(* IEC 61131-3 sources: xPLCCore/codesys_code/Application/COMM_FBs/FB_MsgPakLevelParser, 7 files *)

(* ---- FB_MsgPakLevelParser.st ---- *)
(* ============================================================================
   FB_MsgPakLevelParser

   A state machine-based parser for MessagePack packets that processes data
   byte-by-byte and tracks the nesting level/depth of containers (arrays and maps).

   This parser does NOT decode MessagePack values, only tracks structure depth.
   ============================================================================ *)

FUNCTION_BLOCK FB_MsgPakLevelParser
VAR_INPUT
    in_byte : BYTE;  (* The byte to parse. Call this FB with a new byte for each step. *)
    x_reset : BOOL;  (* Set TRUE to reset the parser state. *)
END_VAR

VAR_OUTPUT
    stk_level_stack : ARRAY[0..29] OF UDINT;  (* Level stack showing remaining elements at each nesting level *)
    ui_level_stack_size : UDINT;              (* Current depth of the stack (number of nested containers) *)
    e_error : E_MsgPakLevelParser_ERROR;      (* Current error code (NONE if no error) *)
END_VAR

VAR
    (* State machine state *)
    e_state : E_MsgPakLevelParser_STATE;

    (* Length accumulation for variable-length types *)
    ui_length_bytes_remaining : UDINT;  (* How many length bytes still needed *)
    ui_length_value : UDINT;             (* Accumulated length value *)
    ui_data_bytes_remaining : UDINT;    (* How many data bytes still needed *)

    (* Track the type byte that caused us to enter EXPECT_LENGTH state *)
    by_last_type_byte : BYTE;  (* Last MessagePack type byte processed *)

    (* Constants *)
    c_MSGPACK_STACK_SIZE : UDINT := 30;  (* Maximum nesting depth *)

    (* Temporary variables *)
    by_current_byte : BYTE;
END_VAR
(* =========== IMPLEMENTATION =========== *)
(* ============================================================================
   Main State Machine Logic
   ============================================================================ *)

(* Handle reset *)
IF x_reset THEN
    ResetParser();
    RETURN;
END_IF

(* If error already occurred, stop processing *)
IF e_error <> E_MsgPakLevelParser_ERROR.NONE THEN
    RETURN;
END_IF

by_current_byte := in_byte;

CASE e_state OF
    E_MsgPakLevelParser_STATE.EXPECT_HEADER:
        (* Process MessagePack type byte *)
        HandleHeaderByte();

    E_MsgPakLevelParser_STATE.EXPECT_LENGTH:
        (* Accumulate length bytes *)
        ProcessLengthBytes();

    E_MsgPakLevelParser_STATE.EXPECT_EXT_TYPE:
        (* Consume extension type byte - no action needed, just transition *)
        e_state := E_MsgPakLevelParser_STATE.EXPECT_DATA;

    E_MsgPakLevelParser_STATE.EXPECT_DATA:
        (* Consume data bytes *)
        ProcessDataBytes();

    ELSE
        e_error := E_MsgPakLevelParser_ERROR.INVALID_STATE;
END_CASE

(* ---- DecrementStack.st ---- *)
METHOD DecrementStack : BOOL
VAR_INPUT
END_VAR
(* =========== IMPLEMENTATION =========== *)

(* Recursively decrement and pop completed levels *)
WHILE ui_level_stack_size > 0 DO
    (* Decrement current level *)
    IF stk_level_stack[ui_level_stack_size - 1] > 0 THEN
        stk_level_stack[ui_level_stack_size - 1] := stk_level_stack[ui_level_stack_size - 1] - 1;
    END_IF

    (* If items still remain in this container, we are done *)
    IF stk_level_stack[ui_level_stack_size - 1] > 0 THEN
        EXIT;
    END_IF

    (* If zero, pop this level and continue to decrement parent *)
    ui_level_stack_size := ui_level_stack_size - 1;
END_WHILE

(* ---- HandleHeaderByte.st ---- *)
METHOD HandleHeaderByte : INT
VAR_INPUT
END_VAR
VAR
    by_type : BYTE;
    ui_count : UDINT;
END_VAR
(* =========== IMPLEMENTATION =========== *)

by_type := by_current_byte;

(* Optimized: Check most common types first (FixInt covers ~50% of all values) *)
(* FixInt: positive (0x00-0x7F) and negative (0xE0-0xFF) *)
IF (by_type <= 16#7F) OR (by_type >= 16#E0) THEN
    DecrementStack();
    e_state := E_MsgPakLevelParser_STATE.EXPECT_HEADER;
    RETURN;
END_IF

(* FixMap (0x80-0x8F: 0-15 pairs) - common container type *)
IF (by_type >= 16#80) AND (by_type <= 16#8F) THEN
    ui_count := by_type - 16#80;
    IF ui_count > 0 THEN
        PushStack(ui_count * 2);
    ELSE
        DecrementStack();
    END_IF
    e_state := E_MsgPakLevelParser_STATE.EXPECT_HEADER;
    RETURN;
END_IF

(* FixArray (0x90-0x9F: 0-15 elements) - common container type *)
IF (by_type >= 16#90) AND (by_type <= 16#9F) THEN
    ui_count := by_type - 16#90;
    IF ui_count > 0 THEN
        PushStack(ui_count);
    ELSE
        DecrementStack();
    END_IF
    e_state := E_MsgPakLevelParser_STATE.EXPECT_HEADER;
    RETURN;
END_IF

(* FixStr (0xA0-0xBF: 0-31 bytes) - common string type *)
IF (by_type >= 16#A0) AND (by_type <= 16#BF) THEN
    ui_count := by_type - 16#A0;
    IF ui_count > 0 THEN
        ui_data_bytes_remaining := ui_count;
        e_state := E_MsgPakLevelParser_STATE.EXPECT_DATA;
    ELSE
        DecrementStack();
        e_state := E_MsgPakLevelParser_STATE.EXPECT_HEADER;
    END_IF
    RETURN;
END_IF

(* Use CASE for exact byte matches - more efficient than IF chain *)
CASE by_type OF
    16#C0:  (* nil *)
        DecrementStack();
        e_state := E_MsgPakLevelParser_STATE.EXPECT_HEADER;

    16#C2:  (* false *)
        DecrementStack();
        e_state := E_MsgPakLevelParser_STATE.EXPECT_HEADER;

    16#C3:  (* true *)
        DecrementStack();
        e_state := E_MsgPakLevelParser_STATE.EXPECT_HEADER;

    16#C4:  (* bin 8 *)
        by_last_type_byte := by_type;
        ui_length_bytes_remaining := 1;
        ui_length_value := 0;
        e_state := E_MsgPakLevelParser_STATE.EXPECT_LENGTH;

    16#C5:  (* bin 16 *)
        by_last_type_byte := by_type;
        ui_length_bytes_remaining := 2;
        ui_length_value := 0;
        e_state := E_MsgPakLevelParser_STATE.EXPECT_LENGTH;

    16#C6:  (* bin 32 *)
        by_last_type_byte := by_type;
        ui_length_bytes_remaining := 4;
        ui_length_value := 0;
        e_state := E_MsgPakLevelParser_STATE.EXPECT_LENGTH;

    16#C7:  (* ext 8 *)
        by_last_type_byte := by_type;
        ui_length_bytes_remaining := 1;
        ui_length_value := 0;
        e_state := E_MsgPakLevelParser_STATE.EXPECT_LENGTH;

    16#C8:  (* ext 16 *)
        by_last_type_byte := by_type;
        ui_length_bytes_remaining := 2;
        ui_length_value := 0;
        e_state := E_MsgPakLevelParser_STATE.EXPECT_LENGTH;

    16#C9:  (* ext 32 *)
        by_last_type_byte := by_type;
        ui_length_bytes_remaining := 4;
        ui_length_value := 0;
        e_state := E_MsgPakLevelParser_STATE.EXPECT_LENGTH;

    16#CA:  (* float 32 *)
        ui_data_bytes_remaining := 4;
        e_state := E_MsgPakLevelParser_STATE.EXPECT_DATA;

    16#CB:  (* float 64 *)
        ui_data_bytes_remaining := 8;
        e_state := E_MsgPakLevelParser_STATE.EXPECT_DATA;

    16#CC:  (* uint 8 *)
        ui_data_bytes_remaining := 1;
        e_state := E_MsgPakLevelParser_STATE.EXPECT_DATA;

    16#CD:  (* uint 16 *)
        ui_data_bytes_remaining := 2;
        e_state := E_MsgPakLevelParser_STATE.EXPECT_DATA;

    16#CE:  (* uint 32 *)
        ui_data_bytes_remaining := 4;
        e_state := E_MsgPakLevelParser_STATE.EXPECT_DATA;

    16#CF:  (* uint 64 *)
        ui_data_bytes_remaining := 8;
        e_state := E_MsgPakLevelParser_STATE.EXPECT_DATA;

    16#D0:  (* int 8 *)
        ui_data_bytes_remaining := 1;
        e_state := E_MsgPakLevelParser_STATE.EXPECT_DATA;

    16#D1:  (* int 16 *)
        ui_data_bytes_remaining := 2;
        e_state := E_MsgPakLevelParser_STATE.EXPECT_DATA;

    16#D2:  (* int 32 *)
        ui_data_bytes_remaining := 4;
        e_state := E_MsgPakLevelParser_STATE.EXPECT_DATA;

    16#D3:  (* int 64 *)
        ui_data_bytes_remaining := 8;
        e_state := E_MsgPakLevelParser_STATE.EXPECT_DATA;

    16#D4:  (* fixext 1 *)
        by_last_type_byte := by_type;
        ui_data_bytes_remaining := 1;
        e_state := E_MsgPakLevelParser_STATE.EXPECT_EXT_TYPE;

    16#D5:  (* fixext 2 *)
        by_last_type_byte := by_type;
        ui_data_bytes_remaining := 2;
        e_state := E_MsgPakLevelParser_STATE.EXPECT_EXT_TYPE;

    16#D6:  (* fixext 4 *)
        by_last_type_byte := by_type;
        ui_data_bytes_remaining := 4;
        e_state := E_MsgPakLevelParser_STATE.EXPECT_EXT_TYPE;

    16#D7:  (* fixext 8 *)
        by_last_type_byte := by_type;
        ui_data_bytes_remaining := 8;
        e_state := E_MsgPakLevelParser_STATE.EXPECT_EXT_TYPE;

    16#D8:  (* fixext 16 *)
        by_last_type_byte := by_type;
        ui_data_bytes_remaining := 16;
        e_state := E_MsgPakLevelParser_STATE.EXPECT_EXT_TYPE;

    16#D9:  (* str 8 *)
        by_last_type_byte := by_type;
        ui_length_bytes_remaining := 1;
        ui_length_value := 0;
        e_state := E_MsgPakLevelParser_STATE.EXPECT_LENGTH;

    16#DA:  (* str 16 *)
        by_last_type_byte := by_type;
        ui_length_bytes_remaining := 2;
        ui_length_value := 0;
        e_state := E_MsgPakLevelParser_STATE.EXPECT_LENGTH;

    16#DB:  (* str 32 *)
        by_last_type_byte := by_type;
        ui_length_bytes_remaining := 4;
        ui_length_value := 0;
        e_state := E_MsgPakLevelParser_STATE.EXPECT_LENGTH;

    16#DC:  (* array 16 *)
        by_last_type_byte := by_type;
        ui_length_bytes_remaining := 2;
        ui_length_value := 0;
        e_state := E_MsgPakLevelParser_STATE.EXPECT_LENGTH;

    16#DD:  (* array 32 *)
        by_last_type_byte := by_type;
        ui_length_bytes_remaining := 4;
        ui_length_value := 0;
        e_state := E_MsgPakLevelParser_STATE.EXPECT_LENGTH;

    16#DE:  (* map 16 *)
        by_last_type_byte := by_type;
        ui_length_bytes_remaining := 2;
        ui_length_value := 0;
        e_state := E_MsgPakLevelParser_STATE.EXPECT_LENGTH;

    16#DF:  (* map 32 *)
        by_last_type_byte := by_type;
        ui_length_bytes_remaining := 4;
        ui_length_value := 0;
        e_state := E_MsgPakLevelParser_STATE.EXPECT_LENGTH;

    ELSE
        (* Invalid byte - not a valid MessagePack type *)
        e_error := E_MsgPakLevelParser_ERROR.UNEXPECTED_BYTE;
END_CASE

(* ---- ProcessDataBytes.st ---- *)
METHOD ProcessDataBytes : BOOL
VAR_INPUT
END_VAR
(* =========== IMPLEMENTATION =========== *)

(* Optimized: combine decrement and check *)
ui_data_bytes_remaining := ui_data_bytes_remaining - 1;

IF ui_data_bytes_remaining = 0 THEN
    (* Data complete *)
    DecrementStack();
    e_state := E_MsgPakLevelParser_STATE.EXPECT_HEADER;
END_IF

(* ---- ProcessLengthBytes.st ---- *)
METHOD ProcessLengthBytes : BOOL
VAR_INPUT
END_VAR
VAR
    ui_shift : UDINT;
END_VAR

(* =========== IMPLEMENTATION =========== *)

(* Accumulate length bytes in big-endian format *)
ui_shift := (ui_length_bytes_remaining - 1) * 8;
ui_length_value := ui_length_value OR (SHL(TO_UDINT(by_current_byte), ui_shift));
ui_length_bytes_remaining := ui_length_bytes_remaining - 1;

IF ui_length_bytes_remaining = 0 THEN
    (* Length complete - optimized type dispatch *)
    (* Check for arrays first *)
    IF (by_last_type_byte = 16#DC) OR (by_last_type_byte = 16#DD) THEN
        (* Array 16 or Array 32 *)
        IF ui_length_value > 0 THEN
            PushStack(ui_length_value);
        ELSE
            DecrementStack();
        END_IF
        e_state := E_MsgPakLevelParser_STATE.EXPECT_HEADER;
    ELSIF (by_last_type_byte = 16#DE) OR (by_last_type_byte = 16#DF) THEN
        (* Map 16 or Map 32 *)
        IF ui_length_value > 0 THEN
            PushStack(ui_length_value * 2);
        ELSE
            DecrementStack();
        END_IF
        e_state := E_MsgPakLevelParser_STATE.EXPECT_HEADER;
    ELSIF (by_last_type_byte = 16#C7) OR (by_last_type_byte = 16#C8) OR (by_last_type_byte = 16#C9) THEN
        (* Ext 8/16/32 *)
        e_state := E_MsgPakLevelParser_STATE.EXPECT_EXT_TYPE;
        ui_data_bytes_remaining := ui_length_value;
    ELSE
        (* String or binary (C4, C5, C6, D9, DA, DB) *)
        ui_data_bytes_remaining := ui_length_value;
        IF ui_data_bytes_remaining > 0 THEN
            e_state := E_MsgPakLevelParser_STATE.EXPECT_DATA;
        ELSE
            (* Empty string/binary *)
            DecrementStack();
            e_state := E_MsgPakLevelParser_STATE.EXPECT_HEADER;
        END_IF
    END_IF
END_IF

(* ---- PushStack.st ---- *)
METHOD PushStack : BOOL
VAR_INPUT
    ui_count : UDINT;  (* Number of elements to push *)
END_VAR
VAR
END_VAR
(* =========== IMPLEMENTATION =========== *)
IF ui_level_stack_size >= c_MSGPACK_STACK_SIZE THEN
    e_error := E_MsgPakLevelParser_ERROR.STACK_OVERFLOW;
    RETURN;
END_IF

stk_level_stack[ui_level_stack_size] := ui_count;
ui_level_stack_size := ui_level_stack_size + 1;

(* ---- ResetParser.st ---- *)
METHOD ResetParser : BOOL
VAR_INPUT
END_VAR
(* =========== IMPLEMENTATION =========== *)
(* Reset state machine *)
e_state := E_MsgPakLevelParser_STATE.EXPECT_HEADER;

(* Reset stack *)
ui_level_stack_size := 0;

(* Reset length accumulation *)
ui_length_bytes_remaining := 0;
ui_length_value := 0;
ui_data_bytes_remaining := 0;

(* Reset type tracking *)
by_last_type_byte := 0;

(* Reset error *)
e_error := E_MsgPakLevelParser_ERROR.NONE;
